TYPE InputBase_8311D824 :
STRUCT
END_STRUCT
END_TYPE

(* stored: Version 1.1.0.1, ProductVersion 3.1.4024.9
   DUT InputBase_8311D824: Id {c891157b-3f1d-424f-9713-bd76cbd8dcae} *)
